PROGRAM testFlexiBuffer
VAR
	shelf : Shelf(2, 2);
	shelfElements: ARRAY[0..100] OF ShelfElement;
	
	flexibuf: FlexiBuffer;
	state: ETestFlexiBufferState;
	
	shelfElement: IShelfElement;
	
	usedElementsCount: UINT := 0;
	i: UINT;
END_VAR


shelf.getNextFreeSpace();

CASE state OF
ETestFlexiBufferState.INIT:
	FOR i:=0 TO 3 DO
		usedElementsCount := usedElementsCount + 1;
		flexibuf.addElement(shelfElements[usedElementsCount - 1]);
	END_FOR;
	state := ETestFlexiBufferState.WAIT;
	
ETestFlexiBufferState.ADD_ELEMENT:
	usedElementsCount := usedElementsCount + 1;	
	flexibuf.addElement(shelfElements[usedElementsCount-1]);	
	state := ETestFlexiBufferState.WAIT;

ETestFlexiBufferState.REMOVE_ELEMENT:
	shelfElement := flexibuf.removeFirstElement();
	state := ETestFlexiBufferState.WAIT;
	
END_CASE

END_PROGRAM

(* stored: Version 1.1.0.1
   POU testFlexiBuffer: Id {9bf03d54-e4de-47fd-9738-beea5cb57baa}, SpecialFunc None *)
